FUNCTION_BLOCK CentralServer (* Basic Function Block Type *)
  (* Standard: 61499-2 *)
  (* Version 0.2, 2003-12-04, JHC, Rockwell Automation, Renamed for better indexing. *)
  (* Version 0.1, 2002-11-05, JHC, Rockwell Automation, Corrected missing ST element in Algorithm REQ. *)
  (* Version 0.0, 2000-05-30, JHC, Rockwell Automation *)
  (* Compiler header: package fb.rt.template; *)
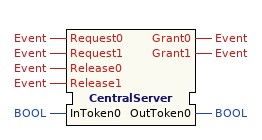
  EVENT_INPUT
    Request0; (* Initialization Request *)
    Request1; (* dab *)
    Release0;
    Release1;
  END_EVENT
  EVENT_OUTPUT
    Grant0; (* Initialization Confirm *)
    Grant1; (* Execution Confirmation *)
  END_EVENT
  VAR_INPUT
    InToken0 : BOOL; (* Input event qualifier *)
  END_VAR
  VAR_OUTPUT
    OutToken0 : BOOL; (* Output event qualifier *)
  END_VAR
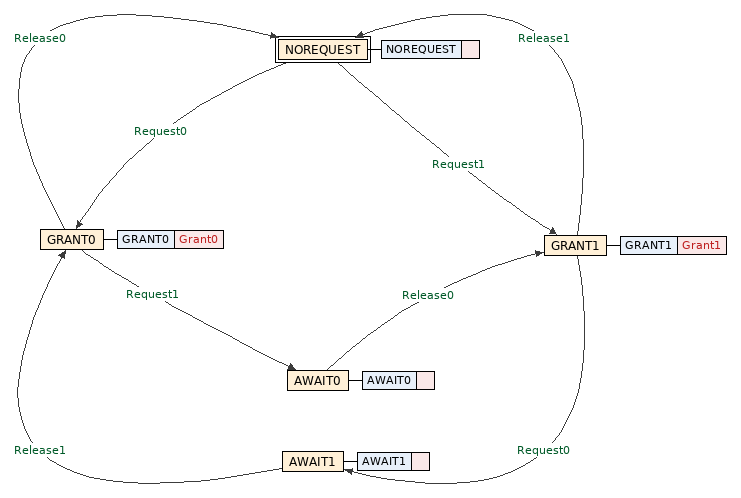
  EC_STATES
    NOREQUEST : NOREQUEST; (* Init state *)
    GRANT0 : GRANT0 -> Grant0;
    GRANT1 : GRANT1 -> Grant1;
    AWAIT0 : AWAIT0;
    AWAIT1 : AWAIT1;
  END_STATES
  EC_TRANSITIONS
    NOREQUEST TO GRANT0 := Request0;
    GRANT0 TO NOREQUEST := Release0;
    NOREQUEST TO GRANT1 := Request1;
    GRANT1 TO NOREQUEST := Release1;
    GRANT0 TO AWAIT0 := Request1;
    AWAIT0 TO GRANT1 := Release0;
    GRANT1 TO AWAIT1 := Request0;
    AWAIT1 TO GRANT0 := Release1;
  END_TRANSITIONS
  ALGORITHM GRANT0 IN Java: (* Initialization algorithm *)
System.out.println("Token Granted to 0");
  END_ALGORITHM
  ALGORITHM GRANT1 IN Java: (* Initialization algorithm *)
System.out.println("Token Granted to 1");
  END_ALGORITHM
  ALGORITHM NOREQUEST IN Java: (* Normally executed algorithm *)
System.out.println("No request");
  END_ALGORITHM
  ALGORITHM AWAIT0 IN Java: (* Normally executed algorithm *)
System.out.println("Awaiting 0");
  END_ALGORITHM
  ALGORITHM AWAIT1 IN Java: (* Normally executed algorithm *)
System.out.println("Await 1");
  END_ALGORITHM
END_FUNCTION_BLOCK
